ABB RAPID module: testmodule.modx

MODULE testmodule

    PROC TestProc()
        TPWrite "hello";
    ENDPROC

ENDMODULE
